FUNCTION_BLOCK FB_SVs
VAR_IN_OUT

END_VAR
VAR_INPUT
	Freigabe_auto			: BOOL;
	Freigabe_Deakt_auto		: BOOL;
	Stellung_Anford_auto	: BOOL;
	Quittierung				: BOOL;
	Parameter_init			: ST_SV_Parameter;
END_VAR
VAR_OUTPUT
	{attribute 'OPC.UA.DA' := '1'}Parameter				: ST_SV_Parameter;			
	{attribute 'OPC.UA.DA' := '1'}Steuerung				: ST_SV_Steuerung;			
	{attribute 'OPC.UA.DA' := '1'}Stellwert				: ST_SV_Stellwert;			
	{attribute 'OPC.UA.DA' := '1'}Zustand					: ST_SVs_Zustand;		

END_VAR
VAR
	Zustandscheck			: FB_SVs_Zustandscheck;
	Logik					: FB_SVs_Logik;
	Ablaufsteuerung			: FB_SVs_Ablaufsteuerung;
	QuitTrig				: FB_SetResetFallTrigger;

	LeseDaten				: FB_SVs_Input;

	IN_Zustand_Stellungrueckmeldung0 		AT %I* : BOOL;
	IN_Zustand_Stellungrueckmeldung1 		AT %I* : BOOL;

	SchreibeDaten			: FB_SVs_Output;
	OUT_Stellung				AT %Q* : BOOL;

END_VAR

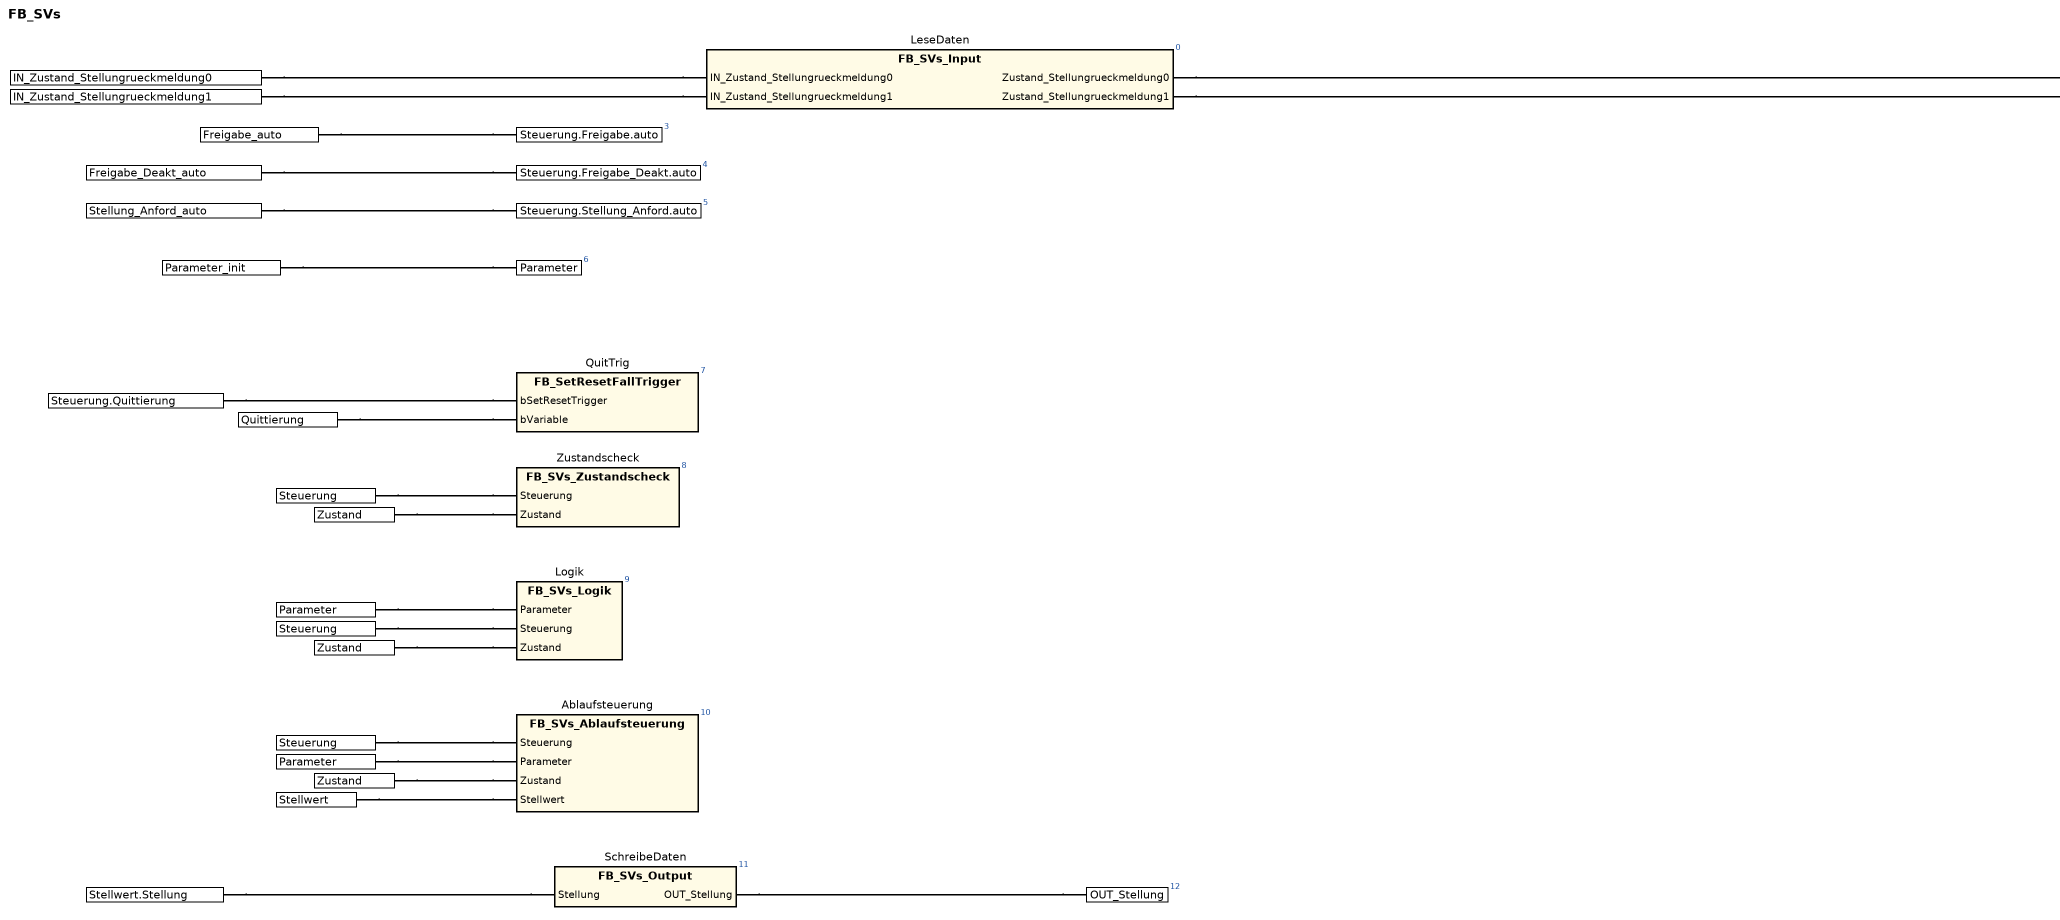
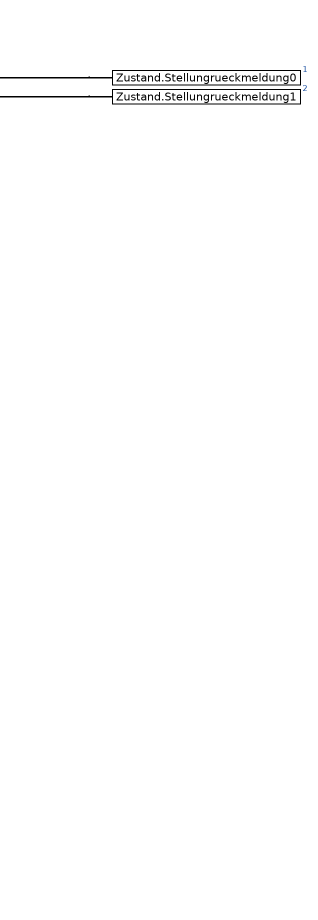
LeseDaten(IN_Zustand_Stellungrueckmeldung0 := IN_Zustand_Stellungrueckmeldung0, IN_Zustand_Stellungrueckmeldung1 := IN_Zustand_Stellungrueckmeldung1); // FB_SVs_Input
Zustand.Stellungrueckmeldung0 := LeseDaten.Zustand_Stellungrueckmeldung0;
Zustand.Stellungrueckmeldung1 := LeseDaten.Zustand_Stellungrueckmeldung1;
Steuerung.Freigabe.auto := Freigabe_auto;
Steuerung.Freigabe_Deakt.auto := Freigabe_Deakt_auto;
Steuerung.Stellung_Anford.auto := Stellung_Anford_auto;
Parameter := Parameter_init;
QuitTrig(bSetResetTrigger := Steuerung.Quittierung, bVariable := Quittierung); // FB_SetResetFallTrigger
Zustandscheck(Steuerung := Steuerung, Zustand := Zustand); // FB_SVs_Zustandscheck
Logik(Parameter := Parameter, Steuerung := Steuerung, Zustand := Zustand); // FB_SVs_Logik
Ablaufsteuerung(Steuerung := Steuerung, Parameter := Parameter, Zustand := Zustand, Stellwert := Stellwert); // FB_SVs_Ablaufsteuerung
SchreibeDaten(Stellung := Stellwert.Stellung); // FB_SVs_Output
OUT_Stellung := SchreibeDaten.OUT_Stellung;

END_FUNCTION_BLOCK

(* stored: Version 1.1.0.1, ProductVersion 3.1.4024.9
   POU FB_SVs: Id {a542d9d8-76dc-405e-965c-a82958b00c8b}, SpecialFunc None *)
